{attribute 'qualified_only'}
{attribute 'strict'}
TYPE E_SortedOrder :
(
	Id,
	Value,
	Duration
);
END_TYPE

(* stored: Version 1.1.0.1, ProductVersion 3.1.4024.12
   DUT E_SortedOrder: Id {a21b9025-e3bf-4802-a4be-122a7f5e7dd2} *)
